# EPICS autosave request: pointGreyApp/Db/pointGrey_settings.req
$(P)$(R)VideoMode
$(P)$(R)Format7Mode
$(P)$(R)FrameRate
$(P)$(R)PixelFormat
$(P)$(R)BinningMode
$(P)$(R)PacketSize
$(P)$(R)PacketDelay
$(P)$(R)ConvertPixelFormat
$(P)$(R)TriggerSource
$(P)$(R)TriggerPolarity
$(P)$(R)SkipFrames
$(P)$(R)StrobeSource
$(P)$(R)StrobeEnable
$(P)$(R)StrobePolarity
$(P)$(R)StrobeDelay
$(P)$(R)StrobeDuration
